// TwinCAT 3 PLC project Test_PLC
// ProgramVersion: 3.1.4023.0
// libraries:
//   Tc2_Standard, * (Beckhoff Automation GmbH)
//   Tc2_System, * (Beckhoff Automation GmbH)
//   Tc3_Module, * (Beckhoff Automation GmbH)
// project tree:
//   / PlcTask.TcTTO
//   POUs/ FB_Test.TcPOU, MAIN.TcPOU
// real-time tasks:
//   TASK PlcTask: cycle T#10ms, priority 20, ADS port 350

CONFIGURATION Test_PLC
    RESOURCE PLC ON TwinCAT3
        TASK PlcTask(INTERVAL := T#10ms, PRIORITY := 21);
        PROGRAM MAIN WITH PlcTask : MAIN;
    END_RESOURCE
END_CONFIGURATION

// ---- POUs/MAIN.TcPOU
PROGRAM MAIN
VAR
	fbTest : FB_Test;
	
	i : INT;
	
	nTest : INT;
END_VAR

fbTest();

CASE i OF
	1: fbTest();
	
	2: fbTest(); nTest := fbTest.iRes;
END_CASE

END_PROGRAM

// ---- POUs/FB_Test.TcPOU
FUNCTION_BLOCK FB_Test
VAR_INPUT
END_VAR
VAR_OUTPUT
	iRes : INT;
END_VAR
VAR
		nMode : BYTE := 0;
		b0 : BIT;
		b1 : BIT;
		b2 : BIT;
	
END_VAR


nMode.0 := b0;
nMode.1 := b1;
nMode.2 := b2;

iRes := nMode;

END_FUNCTION_BLOCK
